{attribute addProperty BoxType "EL2521-1001-0000"}
{attribute addProperty Id "InputsAT %I*Inputs_44EC503A2430OutputsAT %Q*Outputs_C13D2F242430WcStateAT %I*WcState_F855686C1620InfoDataAT %I*InfoData_BC63D37F80100"}
{attribute addProperty CRC "1350076304"}
{attribute addProperty SizeInBites "144"}
{attribute addProperty SizeInBytes "18"}
TYPE EL2521_47043442 :
STRUCT
	{attribute addProperty Name "Inputs"}
	Inputs : Inputs_44EC503A;
	{attribute addProperty Name "Outputs"}
	Outputs : Outputs_C13D2F24;
	{attribute addProperty Name "WcState"}
	WcState : WcState_F855686C;
	{attribute addProperty Name "InfoData"}
	InfoData : InfoData_BC63D37F;
END_STRUCT
END_TYPE

(* stored: Version 1.2.0.0, ProductVersion 3.1.4024.9
   DUT EL2521_47043442: Id {3d460e96-320a-4b79-9e76-a2c2328df7be} *)
